FUNCTION_BLOCK FB_System_BWK_Ablaufsteuerung
VAR_IN_OUT
	Zustand				: ST_System_BWK_Zustand;
	Stellwert			: ST_System_BWK_Stellwert;
	Steuerung			: ST_System_BWK_Steuerung;
END_VAR
VAR_INPUT
	Zustand_Stellventil		: ST_SV_Zustand;
	Zustand_BWK			: ST_BWK_Zustand;
END_VAR
VAR_OUTPUT
END_VAR
VAR
END_VAR

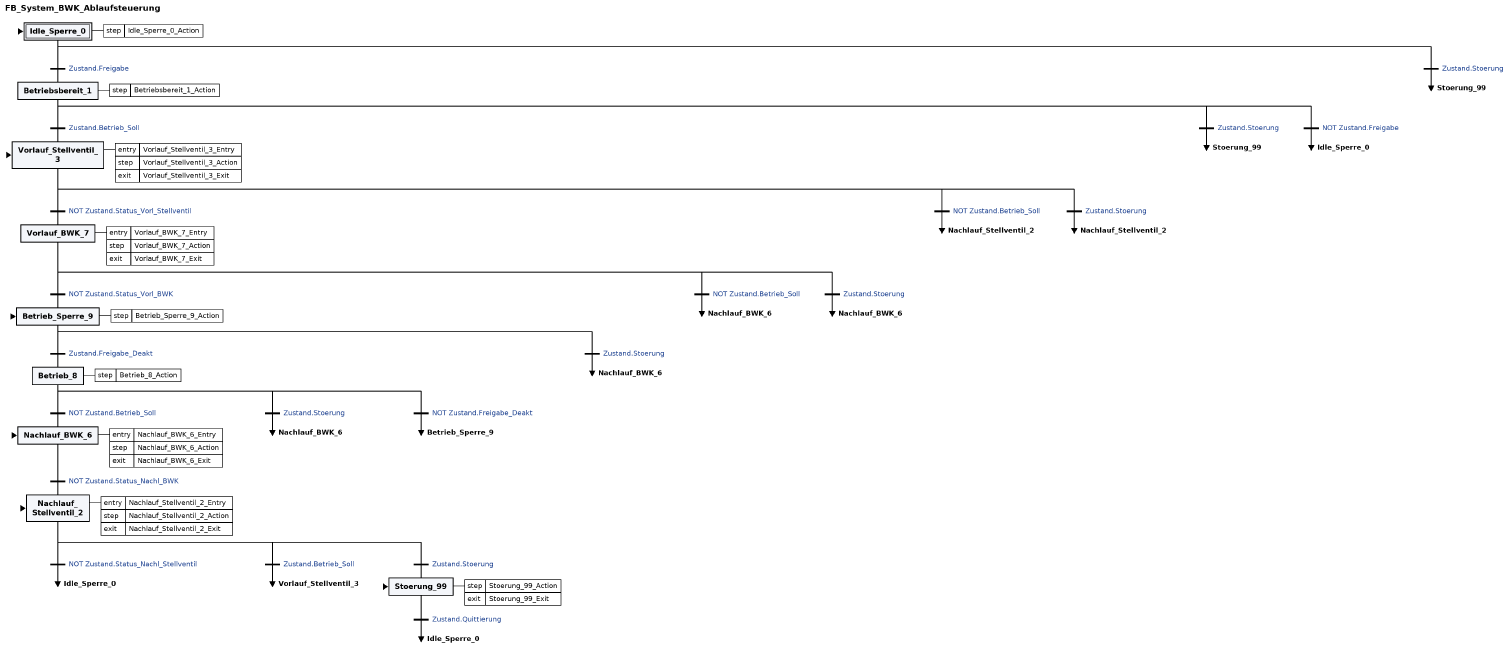
INITIAL_STEP Idle_Sperre_0:
    Idle_Sperre_0_Action(N);  // step action
END_STEP
TRANSITION FROM Idle_Sperre_0 TO Betriebsbereit_1
    := Zustand.Freigabe;
END_TRANSITION
TRANSITION FROM Idle_Sperre_0 TO Stoerung_99
    := Zustand.Stoerung;
END_TRANSITION
STEP Betriebsbereit_1:
    Betriebsbereit_1_Action(N);  // step action
END_STEP
TRANSITION FROM Betriebsbereit_1 TO Vorlauf_Stellventil_3
    := Zustand.Betrieb_Soll;
END_TRANSITION
TRANSITION FROM Betriebsbereit_1 TO Stoerung_99
    := Zustand.Stoerung;
END_TRANSITION
TRANSITION FROM Betriebsbereit_1 TO Idle_Sperre_0
    := NOT Zustand.Freigabe;
END_TRANSITION
STEP Vorlauf_Stellventil_3:
    Vorlauf_Stellventil_3_Entry(P1);  // entry action
    Vorlauf_Stellventil_3_Action(N);  // step action
    Vorlauf_Stellventil_3_Exit(P0);  // exit action
END_STEP
TRANSITION FROM Vorlauf_Stellventil_3 TO Vorlauf_BWK_7
    := NOT Zustand.Status_Vorl_Stellventil;
END_TRANSITION
TRANSITION FROM Vorlauf_Stellventil_3 TO Nachlauf_Stellventil_2
    := NOT Zustand.Betrieb_Soll;
END_TRANSITION
TRANSITION FROM Vorlauf_Stellventil_3 TO Nachlauf_Stellventil_2
    := Zustand.Stoerung;
END_TRANSITION
STEP Vorlauf_BWK_7:
    Vorlauf_BWK_7_Entry(P1);  // entry action
    Vorlauf_BWK_7_Action(N);  // step action
    Vorlauf_BWK_7_Exit(P0);  // exit action
END_STEP
TRANSITION FROM Vorlauf_BWK_7 TO Betrieb_Sperre_9
    := NOT Zustand.Status_Vorl_BWK;
END_TRANSITION
TRANSITION FROM Vorlauf_BWK_7 TO Nachlauf_BWK_6
    := NOT Zustand.Betrieb_Soll;
END_TRANSITION
TRANSITION FROM Vorlauf_BWK_7 TO Nachlauf_BWK_6
    := Zustand.Stoerung;
END_TRANSITION
STEP Betrieb_Sperre_9:
    Betrieb_Sperre_9_Action(N);  // step action
END_STEP
TRANSITION FROM Betrieb_Sperre_9 TO Betrieb_8
    := Zustand.Freigabe_Deakt;
END_TRANSITION
TRANSITION FROM Betrieb_Sperre_9 TO Nachlauf_BWK_6
    := Zustand.Stoerung;
END_TRANSITION
STEP Betrieb_8:
    Betrieb_8_Action(N);  // step action
END_STEP
TRANSITION FROM Betrieb_8 TO Nachlauf_BWK_6
    := NOT Zustand.Betrieb_Soll;
END_TRANSITION
TRANSITION FROM Betrieb_8 TO Nachlauf_BWK_6
    := Zustand.Stoerung;
END_TRANSITION
TRANSITION FROM Betrieb_8 TO Betrieb_Sperre_9
    := NOT Zustand.Freigabe_Deakt;
END_TRANSITION
STEP Nachlauf_BWK_6:
    Nachlauf_BWK_6_Entry(P1);  // entry action
    Nachlauf_BWK_6_Action(N);  // step action
    Nachlauf_BWK_6_Exit(P0);  // exit action
END_STEP
TRANSITION FROM Nachlauf_BWK_6 TO Nachlauf_Stellventil_2
    := NOT Zustand.Status_Nachl_BWK;
END_TRANSITION
STEP Nachlauf_Stellventil_2:
    Nachlauf_Stellventil_2_Entry(P1);  // entry action
    Nachlauf_Stellventil_2_Action(N);  // step action
    Nachlauf_Stellventil_2_Exit(P0);  // exit action
END_STEP
TRANSITION FROM Nachlauf_Stellventil_2 TO Idle_Sperre_0
    := NOT Zustand.Status_Nachl_Stellventil;
END_TRANSITION
TRANSITION FROM Nachlauf_Stellventil_2 TO Vorlauf_Stellventil_3
    := Zustand.Betrieb_Soll;
END_TRANSITION
TRANSITION FROM Nachlauf_Stellventil_2 TO Stoerung_99
    := Zustand.Stoerung;
END_TRANSITION
STEP Stoerung_99:
    Stoerung_99_Action(N);  // step action
    Stoerung_99_Exit(P0);  // exit action
END_STEP
TRANSITION FROM Stoerung_99 TO Idle_Sperre_0
    := Zustand.Quittierung;
END_TRANSITION

ACTION Betrieb_8_Action:
(* Stellwert setzen *)
Stellwert.Anford_Stellventil		:= TRUE;
Stellwert.Anford_BWK			:= TRUE;

(* Zustand setzen *)
Zustand.Status				:= E_System_BWK_Zustand_Status_Betrieb;
END_ACTION

ACTION Betrieb_Sperre_9_Action:
(* Stellwert setzen *)
Stellwert.Anford_Stellventil		:= TRUE;
Stellwert.Anford_BWK		:= TRUE;

(* Zustand setzen *)
Zustand.Status				:= E_System_BWK_Zustand_Status_Betrieb_Sperre;
END_ACTION

ACTION Betriebsbereit_1_Action:
(* Stellwert setzen *)
Stellwert.Anford_Stellventil	:= FALSE;
Stellwert.Anford_BWK	:= FALSE;

(* Zustand setzen *)
Zustand.Status			:= E_System_BWK_Zustand_Status_Betriebsbereit;
END_ACTION

ACTION Idle_Sperre_0_Action:
(* Stellwert setzen *)
Stellwert.Anford_Stellventil	:= FALSE;
Stellwert.Anford_BWK		:= FALSE;

(* Zustand setzen *)
Zustand.Status			:= E_System_BWK_Zustand_Status_Idle_Sperre;


(* Quittierungszustand auf False setzen, damit das System bei einer erneuten Störung nicht direkt wieder angeschaltet wird *)
Steuerung.Quittierung	:= FALSE;
END_ACTION

ACTION Nachlauf_BWK_6_Action:
(* Stellwert setzen *)
Stellwert.Anford_Stellventil		:= TRUE;
Stellwert.Anford_BWK			:= FALSE;

(* Zustand setzen *)
Zustand.Status				:= E_System_BWK_Zustand_Status_Nachl_BWK;
Zustand.Status_Nachl_BWK		:= Zustand_BWK.Betrieb OR Zustand_BWK.Status_Nachl;
END_ACTION

ACTION Nachlauf_BWK_6_Entry:
Zustand.Status_Nachl_BWK		:= TRUE;
END_ACTION

ACTION Nachlauf_BWK_6_Exit:
Zustand.Status_Nachl_BWK		:= FALSE;
END_ACTION

ACTION Nachlauf_Stellventil_2_Action:
(* Stellwert setzen *)
Stellwert.Anford_Stellventil		:= FALSE;
Stellwert.Anford_BWK			:= FALSE;

(* Zustand setzen *)
Zustand.Status				:= E_System_BWK_Zustand_Status_Nachl_Stellventil;
Zustand.Status_Nachl_Stellventil	:= Zustand_Stellventil.Stellung OR Zustand_Stellventil.Stellungwechsel10;
END_ACTION

ACTION Nachlauf_Stellventil_2_Entry:
Zustand.Status_Nachl_Stellventil	:= TRUE;
END_ACTION

ACTION Nachlauf_Stellventil_2_Exit:
Zustand.Status_Nachl_Stellventil	:= FALSE;
END_ACTION

ACTION Stoerung_99_Action:
(* Stellwert setzen *)
Stellwert.Anford_Stellventil	:= FALSE;
Stellwert.Anford_BWK		:= FALSE;

(* Zustand setzen *)
Zustand.Stoerung			:= TRUE;
Zustand.Status			:= E_System_BWK_Zustand_Status_Stoerung;
END_ACTION

ACTION Stoerung_99_Exit:
Zustand.Stoerung	:= FALSE;
END_ACTION

ACTION Vorlauf_BWK_7_Action:
(* Stellwert setzen *)
Stellwert.Anford_Stellventil		:= TRUE;
Stellwert.Anford_BWK			:= TRUE;

(* Zustand setzen *)
Zustand.Status				:= E_System_BWK_Zustand_Status_Vorl_BWK;
Zustand.Status_Vorl_BWK		:= NOT(Zustand_BWK.Betrieb AND NOT Zustand_BWK.Status_Vorl);
END_ACTION

ACTION Vorlauf_BWK_7_Entry:
Zustand.Status_Vorl_BWK		:= TRUE;
END_ACTION

ACTION Vorlauf_BWK_7_Exit:
Zustand.Status_Vorl_BWK		:= FALSE;
END_ACTION

ACTION Vorlauf_Stellventil_3_Action:
(* Stellwert setzen *)
Stellwert.Anford_Stellventil		:= TRUE;
Stellwert.Anford_BWK			:= FALSE;

(* Zustand setzen *)
Zustand.Status				:= E_System_BWK_Zustand_Status_Vorl_Stellventil;
Zustand.Status_Vorl_Stellventil	:= NOT(Zustand_Stellventil.Stellung AND NOT Zustand_Stellventil.Stellungwechsel01);
END_ACTION

ACTION Vorlauf_Stellventil_3_Entry:
Zustand.Status_Vorl_Stellventil	:= TRUE;
END_ACTION

ACTION Vorlauf_Stellventil_3_Exit:
Zustand.Status_Vorl_Stellventil	:= FALSE;
END_ACTION

END_FUNCTION_BLOCK

(* stored: Version 1.1.0.1, ProductVersion 3.1.4024.9
   POU FB_System_BWK_Ablaufsteuerung: Id {5ffd9306-c673-4f0e-a3e6-0dbdc8bbf54b}, SpecialFunc None
   Action Betrieb_8_Action: Id {ab25f02e-90ab-4cdb-888d-7c2d67cbdbfa}
   Action Betrieb_Sperre_9_Action: Id {0223f5ac-ae1f-42b7-ae0d-7dcdb1633022}
   Action Betriebsbereit_1_Action: Id {a7a7a589-f0c5-4aef-aa25-892958eaf117}
   Action Idle_Sperre_0_Action: Id {d55ff16c-2883-495b-8a9c-d40f8d60f6b7}
   Action Nachlauf_BWK_6_Action: Id {c5469d61-b19f-40f8-ab2b-f99091e29236}
   Action Nachlauf_BWK_6_Entry: Id {9fe2115f-0f9b-404f-87db-c2aefd90eda2}
   Action Nachlauf_BWK_6_Exit: Id {0fd6fe68-8ef8-4e96-83cd-b496bb882770}
   Action Nachlauf_Stellventil_2_Action: Id {caedfa0f-2f08-45b1-8b6d-11ba6b4450ea}
   Action Nachlauf_Stellventil_2_Entry: Id {990e2bc2-5651-4fac-9ca7-36a494e002f3}
   Action Nachlauf_Stellventil_2_Exit: Id {e37f0ca1-5437-419b-8732-69df92525dde}
   Action Stoerung_99_Action: Id {6bd567c6-ead5-4ed4-8e1c-c3eb03a275d3}
   Action Stoerung_99_Exit: Id {0778e571-bcc2-483f-a317-e30795c13202}
   Action Vorlauf_BWK_7_Action: Id {b06245d8-023c-4ca0-98e5-0b9eda9da62a}
   Action Vorlauf_BWK_7_Entry: Id {84cf6830-4742-42a6-ad3f-d890742a1de5}
   Action Vorlauf_BWK_7_Exit: Id {38a5e0ee-94db-448c-b533-83cfba7df42a}
   Action Vorlauf_Stellventil_3_Action: Id {d42ad451-3782-4bf8-a020-5c2343523fb8}
   Action Vorlauf_Stellventil_3_Entry: Id {a75351d4-98b0-46c8-a7b2-fd38320e485b}
   Action Vorlauf_Stellventil_3_Exit: Id {5b771e44-612e-4e9f-a261-3f853bdd5c4d} *)
